FUNCTION_BLOCK FB_MotorsPowerUp
VAR_INPUT
	bExecute : BOOL;
END_VAR
VAR_OUTPUT
	bPowerUpError 	: BOOL := FALSE;
	bPowerUpDone 	: BOOL := FALSE;
END_VAR
VAR
	eState    	: (Reset, M1, M2, M3); 
	fbMCPower 	: MC_Power;
		PowerErrorID	: UDINT;
		bPowerStatus	: BOOL := FALSE;
		bM2 : BOOL := FALSE;
		bM3 : BOOL := FALSE;
END_VAR

CASE eState OF
	Reset:
		bPowerUpDone := FALSE;
		eState := M1;
	M1:
		IF bExecute THEN
			fbMcPower(
				Axis 			:= GVL_Motion.M1Motor.Axis,	//axisPointer^,
				Enable 			:= TRUE, 	//Enable the Axis if the driver is ready without safety fauls
				Enable_Positive := TRUE, 	//Enable for positive moviments
				Enable_Negative := TRUE, 	//Enable for negative moviments
				Error			=> bPowerUpError,
				ErrorID			=> PowerErrorID,	 //Error ID if the power enter in error.
				Status			=> bPowerStatus
			);
		END_IF
		IF bPowerStatus THEN
			eState := M2;
			//bPowerUpDone := TRUE;
		END_IF
	M2:
		IF bExecute THEN
			fbMcPower(
				Axis 			:= GVL_Motion.M2Motor.Axis,	//axisPointer^,
				Enable 			:= TRUE, 	//Enable the Axis if the driver is ready without safety fauls
				Enable_Positive := TRUE, 	//Enable for positive moviments
				Enable_Negative := TRUE, 	//Enable for negative moviments
				Error			=> bPowerUpError,
				ErrorID			=> PowerErrorID,	 //Error ID if the power enter in error.
				Status			=> bPowerStatus
			);
		END_IF
		IF bPowerStatus THEN
			eState := M3;
			//bPowerUpDone := TRUE;
		END_IF
	
	M3:
		IF bExecute THEN
			fbMcPower(
				Axis 			:= GVL_Motion.M3Motor.Axis,	//axisPointer^,
				Enable 			:= TRUE, 	//Enable the Axis if the driver is ready without safety fauls
				Enable_Positive := TRUE, 	//Enable for positive moviments
				Enable_Negative := TRUE, 	//Enable for negative moviments
				Error			=> bPowerUpError,
				ErrorID			=> PowerErrorID,	 //Error ID if the power enter in error.
				Status			=> bPowerStatus
			);
		END_IF
		IF bPowerStatus THEN
			bPowerUpDone := TRUE;
		END_IF
	
END_CASE

END_FUNCTION_BLOCK

(* stored: Version 1.1.0.1, ProductVersion 3.1.4024.12
   POU FB_MotorsPowerUp: Id {2ede40b4-9170-4e3a-965e-058f9fe9c946}, SpecialFunc None *)
